// TwinCAT 3 PLC project Untitled1
// ProgramVersion: 3.1.4024.0
// libraries:
//   Tc2_Standard, * (Beckhoff Automation GmbH)
//   Tc2_System, * (Beckhoff Automation GmbH)
//   Tc2_TcpIp, * (Beckhoff Automation GmbH)
//   Tc2_Utilities, * (Beckhoff Automation GmbH)
//   Tc3_Module, * (Beckhoff Automation GmbH)
// project tree:
//   GVLs/ GVL_TCPIP.TcGVL
//   / PlcTask.TcTTO
//   POUs/ MAIN.TcPOU
//   TcpIp/ FB_ClientConnection.TcPOU, FB_FIFO_Frame.TcPOU, FB_FIFO_Log.TcPOU, TcpIp_Client.TcPOU
// real-time tasks:
//   TASK PlcTask: cycle T#10ms, priority 20, ADS port 350

CONFIGURATION Untitled1
    RESOURCE PLC ON TwinCAT3
        TASK PlcTask(INTERVAL := T#10ms, PRIORITY := 20);
        PROGRAM MAIN WITH PlcTask : MAIN;
    END_RESOURCE
END_CONFIGURATION

// ---- GVLs/GVL_TCPIP.TcGVL
VAR_GLOBAL CONSTANT
	PLCPRJ_BUFFER_SIZE						: UDINT := 1000;(* Max. internal fifo/receiver buffer size *)

	(* Some project specific error codes *)
	PLCPRJ_ERROR_RECEIVE_TIMEOUT			: UDINT := 16#8101;(* Receive timeout *)
	PLCPRJ_ERROR_SENDFIFO_OVERFLOW			: UDINT := 16#8102;(* Send fifo overflow *)
	PLCPRJ_ERROR_RECFIFO_OVERFLOW			: UDINT := 16#8103;(* Receive fifo overflow *)
END_VAR

// ---- POUs/MAIN.TcPOU
PROGRAM MAIN
VAR
	fbCloseAll		: FB_SocketCloseAll;
	bInitalized: BOOL;
END_VAR

IF NOT bInitalized THEN
	fbCloseAll(bExecute := TRUE);
ELSE
	Tcpip_Client();
END_IF

IF NOT fbCloseAll.bBusy THEN
	bInitalized := TRUE;
END_IF

END_PROGRAM

// ---- TcpIp/TcpIp_Client.TcPOU
PROGRAM TcpIp_Client
VAR
	ClientConnection : FB_ClientConnection;
	
	fbTx 		: FB_FIFO_Frame('TestTx');(* TX fifo *)
	fbRx 		: FB_FIFO_Frame('TestRx');(* RX fifo *)
	fbLog		: FB_FIFO_Log('TestLog');(* Log message fifo *)
	Timer: TON;
	bEnable: BOOL;
	nPort: UDINT;
	bLoging: BOOL;
	nTest : BYTE;
	nCounter : BYTE;
END_VAR

ClientConnection.isEnabling := bEnable;
ClientConnection.isLogging := bLoging;
ClientConnection.Name := 'Test::';
ClientConnection.ReconnectTime := T#40S;
ClientConnection.RemoteHost := '127.0.0.1';
ClientConnection.RemotePort := nPort;
ClientConnection.Delimiter := nTest;
ClientConnection(fbTx := fbTx, fbRx := fbRx, fbLog := fbLog);

fbTx.isLogging := TRUE;
fbRx.isLogging := TRUE;
fbLog.isLogging := TRUE;

IF ClientConnection.ConnectionState = eSocket_Connected THEN
Timer(IN:=TRUE, PT:=T#1S);	
	IF Timer.Q THEN
		Timer(IN:=FALSE);
		nCounter := nCounter + 1;
		fbTx.AddTail(ConCAT('Hello',BYTE_TO_STRING(nCounter)));
	END_IF
END_IF

END_PROGRAM

// ---- TcpIp/FB_ClientConnection.TcPOU
(* This function block implements simple TCP/IP client protocol. *)
FUNCTION_BLOCK FB_ClientConnection
VAR_IN_OUT
	fbTx 		: FB_FIFO_Frame;(* TX fifo *)
	fbRx 		: FB_FIFO_Frame;(* RX fifo *)
	fbLog		: FB_FIFO_Log;(* Log message fifo *)
END_VAR
VAR
	_sSrvNetID	: T_AmsNetID	:= '';(* TwinCAT TCP/IP server network address *)
	_sRemoteHost	: T_IPv4Addr	:= '127.0.0.1';(* IP address of remote server *)
	_nRemotePort	: UDINT			:= 200;(* Remote server port *)
	_bEnable		: BOOL			:= FALSE;(* TRUE => Enable/connect, FALSE => Disable/disconnect *)
	_tReconnect	: TIME 			:= T#45S;(* Try to reconnect after this time *)
	_bLog		: BOOL 			:= FALSE;(* TRUE => Enable log message output, FALSE => Disable *)
	_sPrefix		: STRING 		:= 'CLIENT::';(* Log message description string (allows the identification of log message source) *)

	_eState		: E_SocketConnectionState := eSOCKET_DISCONNECTED;(* TCP/IP connection state *)

	fbConnect 	: FB_ClientServerConnection;(* Create/release TCP/IP connection *)
	fbSend		: FB_SocketSend;(* Send TCP/IP data *)
	fbReceive	: FB_SocketReceive;(* Receive TCP/IP data *)
	nState 		: BYTE;(* Global state *)
	bSndBusy 	: BOOL;(* Tx state *)
	bRcvBusy 	: BOOL;(* Rx state *)
	bDisconnect	: BOOL;(* Disconnect flag, if set the socket will be closed *)

	fbPollTimer	: TON;(* Receive poll timer *)
	fbResponseTimer	: TON;(* Response timeout timer *)
	fbReconnectTimer : TON;(* Reconnect timer *)

	cbReceived	: UDINT;(* Count of received data bytes *)
	cbRx		: UDINT;(* Byte length of received string *)
	buffer		: ARRAY[0..PLCPRJ_BUFFER_SIZE] OF BYTE;(* Temp. RX buffer *)
	sRxFrame	: T_MaxString;
	sTxFrame	: T_MaxString;
	i			: UDINT;
	bAbort		: BOOL;
	nDelimiter : BYTE := 16#0;
	
END_VAR

VAR CONSTANT
	PLCPRJ_RECEIVE_POLLING_TIME				: TIME := T#100MS;
	PLCPRJ_RECEIVE_TIMEOUT					: TIME := T#50S;
END_VAR

CASE nState OF
	0:(* Connect *)
		fbConnect( 	sSrvNetID 		:= _sSrvNetID,
					nMode			:= SEL( _bLog, 0, CONNECT_MODE_ENABLEDBG),(* Enable/disable debug messages? *)
					sRemoteHost 	:= _sRemoteHost, nRemotePort := _nRemotePort,
					bEnable			:= _bEnable, tReconnect	:= _tReconnect,
					eState			=> _eState );
		IF NOT fbConnect.bBusy THEN
			IF NOT fbConnect.bError THEN
				IF _eState = eSOCKET_CONNECTED THEN(* We are connected *)
					
					fbTx.Clear();(* Clear TX fifo (optional) *)
					fbRx.Clear();(* Clear RX fifo (optional) *)
					fbLog.Clear();(* Clear log fifo (optional) *)
					bSndBusy := FALSE;
					bRcvBusy := FALSE;
					bDisconnect 	:= FALSE;
					cbReceived 		:= 0;

					fbPollTimer( IN := FALSE, PT := T#0S );
					fbResponseTimer( IN := FALSE, PT := PLCPRJ_RECEIVE_TIMEOUT );
					fbReconnectTimer( IN := FALSE, PT := _tReconnect );
				
					fbLog.Message( sMessage := 'Connection established!', hSocket := fbConnect.hSocket );
					nState := 1;
				END_IF
			ELSE(* Connect error => log error *)
				fbLog.Error( sMessage := 'FB_ClientServerConnection()', nErrID := fbConnect.nErrId );
			END_IF
		END_IF


	1:(* Data exchange state *)
		bDisconnect := NOT _bEnable OR bDisconnect;(* User/internal disconnect requested? *)
		IF bDisconnect AND NOT bSndBusy AND NOT bRcvBusy THEN
			bDisconnect := FALSE;
			fbLog.Message( sMessage := 'Closing connection!', hSocket := fbConnect.hSocket );
			nState := 2;(* Disconnect *)
		ELSE

			(* ------------------ Send tx data -------------------------------------- *)
			IF NOT bDisconnect AND NOT bSndBusy THEN
				fbTx.RemoveHead();(* Remove oldest string entry *)
				sTxFrame := fbTx.ReceivedString;
				IF fbTx.isRemovedorAdded THEN(* Success *)
					fbSend( bExecute := FALSE );
					fbSend(	sSrvNetID 	:= _sSrvNetID,
							hSocket		:= fbConnect.hSocket,
							cbLen		:= INT_TO_UDINT(LEN( sTxFrame )) + 1,(* Send string inclusive string (null) delimiter! *)
							pSrc		:= ADR( sTxFrame ),(* Address of the string variable *)
							bExecute	:= TRUE );
					bSndBusy := TRUE;
				END_IF
			ELSE(* Wait until send not busy *)
				fbSend( bExecute := FALSE );
				IF NOT fbSend.bBusy THEN
					bSndBusy := FALSE;
					IF fbSend.bError THEN(* Send error => log error and disconnect *)
						fbLog.Error( sMessage := 'FB_SocketSend()', nErrID := fbSend.nErrId );
						bDisconnect := TRUE;(* Set flag *)
					END_IF
				END_IF
			END_IF
			(* ---------------------------------------------------------------------- *)


			(* ---------------------- Get rx data ----------------------------------- *)
			IF NOT bDisconnect AND NOT bRcvBusy THEN
				
				fbPollTimer( IN := TRUE );
				IF fbPollTimer.Q THEN
					IF fbRx.freeBufferSpace >= SIZEOF(sRxFrame) THEN(* Check free rx fifo space *)
						fbPollTimer( IN := FALSE, PT := PLCPRJ_RECEIVE_POLLING_TIME );
						fbReceive( bExecute := FALSE );
						fbReceive( 	sSrvNetId	:= _sSrvNetID,
									hSocket		:= fbConnect.hSocket,
									cbLen		:= SIZEOF(buffer) - cbReceived,
									pDest		:= ADR(buffer) + cbReceived,
									bExecute	:= TRUE );
						bRcvBusy := TRUE;
					END_IF
				END_IF
				
			ELSE(* Wait until receive not busy *)

				fbReceive( bExecute := FALSE );
				IF NOT fbReceive.bBusy THEN
					bRcvBusy := FALSE;
					IF NOT fbReceive.bError THEN
						IF fbReceive.nRecBytes > 0 THEN(* Bytes received *)
							
							fbPollTimer( IN := FALSE, PT := T#0S );(* Bytes received => increase the read (polling) speed *)
							fbResponseTimer( IN := FALSE );(* Bytes received => disable timeout check *)
							cbReceived := cbReceived + fbReceive.nRecBytes;(* Calculate the number of received data bytes *)

							(* Parse received bytes and extract strings *)
							REPEAT
								bAbort := TRUE;(* set flag *)
								IF cbReceived > 0 THEN

									(* Search for string null delimiter *)
									FOR i:= 0 TO cbReceived - 1 BY 1 DO
										IF buffer[i] = nDelimiter THEN (* End of string position found *)

											cbRx := i + 1;(* Calculate the length of string (inclusive the end delimiter) *)
											MEMCPY( ADR(sRxFrame), ADR(buffer), MIN(cbRx, SIZEOF(sRxFrame) ) );(* Copy string bytes to temp string variable *)

											fbRx.AddTail( sPut := sRxFrame );(* Add string to the rx fifo *)
											IF fbRx.isRemovedorAdded THEN
												MEMMOVE( ADR(buffer), ADR(buffer) + cbRx, cbReceived - cbRx );(* Move/shift remaining bytes in buffer *)
												cbReceived := cbReceived - cbRx;(* Recalculate the remaining data length *)

												IF fbRx.freeBufferSpace >= SIZEOF(sRxFrame) THEN (* Check free rx buffer space *)
													bAbort := FALSE;(* Reset flag, try to parse the next string *)
												END_IF
											ELSE(* Fifo overflow => log error and disconnect *)
												fbLog.Error( sMessage := 'FB_FrameFifo(receiver)', nErrID := PLCPRJ_ERROR_RECFIFO_OVERFLOW );
												bDisconnect := TRUE;(* set flag *)
												RETURN;
											END_IF

											EXIT; (* buffer[i] = 0을 찾으면 Exit *)
										END_IF
									END_FOR

								END_IF (* IF cbReceived > 0 THEN *)

							UNTIL bAbort
							END_REPEAT

						ELSE(* No bytes received *)
							fbResponseTimer( IN := TRUE );(* No bytes received => enable timeout check *)
							IF fbResponseTimer.Q THEN (* Timeout error*)
								fbResponseTimer( IN := FALSE );
								fbLog.Error( sMessage := 'FB_SocketReceive()', nErrID := PLCPRJ_ERROR_RECEIVE_TIMEOUT );
								bDisconnect := TRUE;(* Set flag *)
							END_IF							
						END_IF(* IF fbReceive.nRecBytes > 0 THEN *)
					ELSE(* Receive error => log error and disconnect *)
						fbLog.Error( sMessage := 'FB_SocketReceive()', nErrID := fbReceive.nErrId );
						bDisconnect := TRUE;(* set flag *)
					END_IF
					
				END_IF(* IF NOT fbReceive.bBusy THEN *) 
	
			END_IF(* IF NOT bDisconnect AND NOT bRcvBusy THEN *)
			(* ---------------------------------------------------------------------- *)
			

		END_IF(* IF bDisconnect AND NOT bSndBusy AND NOT bRcvBusy THEN *)


	2:(* Disconnect *)
		fbConnect( bEnable:= FALSE, eState=>_eState );
		IF _eState = eSOCKET_DISCONNECTED THEN
			fbReconnectTimer( IN := TRUE );(* Please wait some seconds and then try to connect again *)
			IF fbReconnectTimer.Q THEN
				fbReconnectTimer( IN := FALSE );
				nState := 0;
			END_IF
		END_IF
END_CASE

PROPERTY ConnectionState : E_SocketConnectionState := eSocket_Disconnected
GET
ConnectionState := _eState;
END_GET
END_PROPERTY

PROPERTY Delimiter : BYTE := 16#1;
GET
Delimiter := nDelimiter;
END_GET
SET
nDelimiter := Delimiter;
END_SET
END_PROPERTY

PROPERTY isEnabling : BOOL := false
GET
isEnabling := _bEnable;
END_GET
SET
_bEnable := isEnabling;
END_SET
END_PROPERTY

PROPERTY isLogging : BOOL
GET
isLogging := _bLog;
END_GET
SET
_bLog := isLogging;
END_SET
END_PROPERTY

PROPERTY Name : STRING
GET
Name := _sPrefix;
END_GET
SET
_sPrefix := Name;
END_SET
END_PROPERTY

PROPERTY ReconnectTime : Time
GET
reconnectTime := _tReconnect;
END_GET
SET
(* ReconnectTime must be morethan 30s *)
IF reconnectTime > T#30S THEN
	_tReconnect := reconnectTime;
ELSE
	reconnectTime := T#31S;
END_IF
END_SET
END_PROPERTY

PROPERTY RemoteHost : T_IPv4Addr
GET
RemoteHost := _sRemoteHost;
END_GET
SET
_sRemoteHost := RemoteHost;
END_SET
END_PROPERTY

PROPERTY RemotePort : UDINT;
GET
RemotePort := _nRemotePort;
END_GET
SET
_nRemotePort := RemotePort;
END_SET
END_PROPERTY

END_FUNCTION_BLOCK

// ---- TcpIp/FB_FIFO_Frame.TcPOU
(* Tx/Rx (string data) fifo control function block *)
FUNCTION_BLOCK FB_FIFO_Frame
VAR
	_Name 					: STRING := ' ';
	_bLog					: BOOL	:= FALSE;(* TRUE => Enable log message output, FALSE => Disable *)
	_bReady					: BOOL;   	(* TRUE = New entry added or removed succesfully, FALSE = Fifo overflow or fifo empty *)
	_numberofString			: UDINT	:= 0;(* Number of fifo entries *)
	_freeBufferSpace		: UDINT := 0;(* Free buffer space *)
	_sGet : T_MAXSTRING;
	
	fbBuffer 	: FB_StringRingBuffer := (bOverwrite := FALSE);(* Basic (lower level) string buffer control function block *)
	buffer		: ARRAY[-3..PLCPRJ_BUFFER_SIZE] OF BYTE;(* Internal buffer memory *)
END_VAR

METHOD AddTail
VAR_INPUT
	sPut		: T_MaxString 	:= '';
END_VAR
fbBuffer.A_AddTail(pBuffer := ADR(Buffer), cbBuffer := SIZEOF(buffer),
				putValue := sPut, bOk => _bReady, nCount => _numberofString);
				
IF _bReady THEN 
	_freeBufferSpace := PLCPRJ_BUFFER_SIZE - fbBuffer.cbSize; (*Calculate the free buffer space*)
	IF _bLog THEN(*Log message*)
		ADSLOGSTR(ADSLOG_MSGTYPE_HINT OR ADSLOG_MSGTYPE_LOG,'%s',sPut);
	END_IF
END_IF
END_METHOD

METHOD Clear
VAR_INPUT
END_VAR
fbBuffer.A_Reset(pBuffer:=ADR(buffer), cbBuffer := SIZEOF(buffer), bOk=>_bReady, getValue => _sGet, nCount => _numberofString );
_freeBufferSpace := PLCPRJ_BUFFER_SIZE;
END_METHOD

METHOD FB_init : BOOL
VAR_INPUT
	bInitRetains : BOOL; // if TRUE, the retain variables are initialized (warm start / cold start)
	bInCopyCode : BOOL;  // if TRUE, the instance afterwards gets moved into the copy code (online change)
	name : STRING;
END_VAR
This^.Name := name;
END_METHOD

PROPERTY FreeBufferSpace : UDINT
GET
freeBufferSpace := _freeBufferSpace;
END_GET
END_PROPERTY

PROPERTY isLogging : BOOL
GET
isLogging := _bLog;
END_GET
SET
_bLog := isLogging;
END_SET
END_PROPERTY

PROPERTY isRemovedorAdded : BOOL
GET
isRemovedorAdded := _bReady;
END_GET
END_PROPERTY

PROPERTY Name : String
GET
Name := _Name;
END_GET
SET
_Name := Name;
END_SET
END_PROPERTY

PROPERTY NumberofString : UDINT
GET
numberofString := _numberofString;
END_GET
END_PROPERTY

PROPERTY ReceivedString : T_MaxString
GET
ReceivedString := _sGet;
END_GET
END_PROPERTY

METHOD RemoveHead
VAR_INPUT
END_VAR
fbBuffer.A_RemoveHead(pBuffer:= ADR(buffer), cbBuffer := SIZEOF(buffer), bOk => _bReady, getValue => _sGet, nCount => _numberofString);

IF _bReady THEN
	_freeBufferSpace := PLCPRJ_BUFFER_SIZE - fbBuffer.cbSize;
END_IF
END_METHOD

END_FUNCTION_BLOCK

// ---- TcpIp/FB_FIFO_Log.TcPOU
(* Log/debug/error message fifo *)
FUNCTION_BLOCK FB_FIFO_Log
VAR
	_bLog		: BOOL 		:= FALSE;(* TRUE => Enable log message output, FALSE => Disable *)
	_Name		: STRING 	:= 'Unknown::';(* Log message description string (allows the identification of log message source) *)
	
	bOk			: BOOL;(* TRUE = New entry added or removed succesfully, FALSE = Fifo overflow or fifo empty *)
	sGet		: T_MaxString := '';(* String entry removed (read) from fifo *)
	nCount		: UDINT := 0;(* Number of fifo entries *)
	fbBuffer 	: FB_StringRingBuffer;(* Basic (lower level) string buffer control function block *)
	buffer		: ARRAY[0..PLCPRJ_BUFFER_SIZE] OF BYTE;(* Internal buffer memory *)
	sSource		: T_MaxString;	
	sPut		: T_MaxString;
END_VAR

;

METHOD Clear : BOOL
VAR_INPUT
END_VAR
(* Clears all fifo entries *)
fbBuffer.A_Reset( 	pBuffer := ADR( buffer ), cbBuffer := SIZEOF( buffer ), 
					bOk=>bOk, nCount=>nCount, getValue=>sGet );
END_METHOD

METHOD Error : BOOL
VAR_INPUT
	sMessage	: STRING 	:= '';(* String message to add (write) to the fifo *)
	nErrID		: UDINT 	:= 0;(* Error code to add (write) to the fifo *)
END_VAR
(* Adds new fifo entry *)
IF nErrID = 0 THEN
	sSource := '::Error: 0x';
ELSIF ( nErrID AND 16#80000000) = 16#80000000 THEN
	IF nErrID = 16#80072746 THEN
		sSource := '::Win32 error (the connection is reset by remote side): 0x';
	ELSE
		sSource := '::Win32 error: 0x';
	END_IF
ELSIF (nErrID AND 16#00008100) = 16#00008100 THEN
	CASE nErrID OF
		PLCPRJ_ERROR_RECEIVE_TIMEOUT:
			sSource := '::PLC sample project receive timeout error: 0x';
		PLCPRJ_ERROR_SENDFIFO_OVERFLOW:
			sSource := '::PLC sample project send fifo overflow error: 0x';
		PLCPRJ_ERROR_RECFIFO_OVERFLOW:
			sSource := '::PLC sample project receive fifo overflow error: 0x';
	ELSE
		sSource := '::Other PLC sample project error: 0x';
	END_CASE
ELSIF (nErrID AND 16#00008000) = 16#00008000 THEN
	sSource := '::Internal TCP/IP Connection Server error: 0x';
ELSE
	sSource := '::TwinCAT System error: 0x';
END_IF

sPut := CONCAT( CONCAT( CONCAT( _name, sMessage ), sSource ), DWORD_TO_HEXSTR( nErrID AND 16#FFFF, 0, FALSE ) ); 

fbBuffer.A_AddTail( pBuffer:= ADR(buffer), cbBuffer:= SIZEOF(buffer),
					putValue:= sPut, bOk=>bOk, nCount=>nCount );
IF bOk THEN
	IF _bLog THEN(* Log error message *)
		ADSLOGSTR( ADSLOG_MSGTYPE_ERROR OR ADSLOG_MSGTYPE_LOG, '%s', sPut );	
	END_IF
END_IF
END_METHOD

METHOD FB_init : BOOL
VAR_INPUT
	bInitRetains : BOOL; // if TRUE, the retain variables are initialized (warm start / cold start)
	bInCopyCode : BOOL;  // if TRUE, the instance afterwards gets moved into the copy code (online change)
	name : STRING;
END_VAR
This^.Name := name;
END_METHOD

PROPERTY isLogging : BOOL
GET
isLogging := _bLog;
END_GET
SET
_bLog := isLogging;
END_SET
END_PROPERTY

METHOD Message : BOOL
VAR_INPUT
	sMessage : STRING;
	hSocket		: T_HSOCKET;(* Socket connection handle *)
END_VAR
(* Adds new fifo entry *)
sPut := CONCAT( CONCAT( _name, sMessage ), CONCAT( '::', HSOCKET_TO_STRING(hSocket) ) );
fbBuffer.A_AddTail( pBuffer:= ADR(buffer), cbBuffer:= SIZEOF(buffer),
					putValue:= sPut, bOk=>bOk, nCount=>nCount );
IF bOk THEN
	IF _bLog THEN(* Log information message *)
		ADSLOGSTR( ADSLOG_MSGTYPE_HINT OR ADSLOG_MSGTYPE_LOG, '%s', sPut );	
	END_IF
END_IF
END_METHOD

PROPERTY Name : String
GET
Name := _Name;
END_GET
SET
_Name := Name;
END_SET
END_PROPERTY

METHOD Remove : BOOL
VAR_INPUT
END_VAR
(* Removes oldest fifo entry *)
IF nCount = 0 THEN
	sGet := '';
	bOk := FALSE;
	RETURN;
END_IF

fbBuffer.A_RemoveHead( pBuffer:= ADR(buffer), cbBuffer:= SIZEOF(buffer),
						getValue=>sGet, bOk=>bOk, nCount=>nCount );
END_METHOD

END_FUNCTION_BLOCK
